# B&R Automation Studio project 8238 (part 9)

#### mnCntCyclic.st - Cyclic code
```iecst
(********************************************************************
 * COPYRIGHT -- Microsoft
 ********************************************************************
 * Program: mnCnt
 * File: mnCntCyclic.st
 * Author: hunholz
 * Created: July 02, 2011
 * Changed: January 3, 2012
 ********************************************************************
 * Implementation of program mnCnt
 ********************************************************************)

PROGRAM _CYCLIC

	/////////////
	// BATCHDATEN
	/////////////

	IF IFmnCnt.In.bBatchEventValid > 0 AND NOT IFmnCnt.Out.xBatchEventReadOK THEN

		// RB Eintrag
		// Jedes Batch-Event wird in den Ringbuffer eingetregen
		IF _xBatchRbOK AND IFmnCnt.In.BatchEvent.bEvent <= MNCNT_BATCHEVENT_DELETE THEN

			_rbBatchIns(pEntry := ADR(IFmnCnt.In.BatchEvent), wPtrWrite := _wPtrWriteBatch, wPtrRead := _wPtrReadBatch, wPtrStart := _wPtrStartBatch);

			IF _rbBatchIns.wStatus <> ERR_OK THEN

				_xBatchRbOK := FALSE;

			END_IF

		END_IF

		// Statistik ergänzen
		// Für jedes Entlade-Event wird ein Gesamtsummenzähler sowie ein Programm-Summenzähler gezählt
		IF _xBatchStatOK AND IFmnCnt.In.BatchEvent.bEvent = MNCNT_BATCHEVENT_UNLOAD THEN

			REPEAT

				_dwBatchStat.enable := TRUE;
				_dwBatchStat.ident := _doBatchStat.ident;
				_dwBatchStat.len := SIZEOF(_lSumWeight);
				_dwBatchStat.pSource := ADR(_lSumWeight);

				IF IFmnCnt.In.BatchEvent.bProgram <= 99 THEN

					// Zunächst die Zähler pro Programm addieren und in das Datenobjekt schreiben. Erst für den 1. Zähler, dann für den 2. Zähler
					_lSumWeight := _BatchStat.Weight1[IFmnCnt.In.BatchEvent.bProgram] + UINT_TO_UDINT(IFmnCnt.In.BatchEvent.Batch.wTotalWeight);

					_dwBatchStat.Offset := ADR(_BatchStat.Weight1[IFmnCnt.In.BatchEvent.bProgram]) - _doBatchStat.pDatObjMem;
					_dwBatchStat();

					IF _dwBatchStat.status <> ERR_OK THEN

						_xBatchStatOK := FALSE;

						EXIT;

					END_IF

					_lSumWeight := _BatchStat.Weight2[IFmnCnt.In.BatchEvent.bProgram] + UINT_TO_UDINT(IFmnCnt.In.BatchEvent.Batch.wTotalWeight);

					_dwBatchStat.Offset := ADR(_BatchStat.Weight2[IFmnCnt.In.BatchEvent.bProgram]) - _doBatchStat.pDatObjMem;
					_dwBatchStat();

					IF _dwBatchStat.status <> ERR_OK THEN

						_xBatchStatOK := FALSE;

						EXIT;

					END_IF

				END_IF

				// Dann wird der Gesamtzähler addiert

				_lSumWeight := _BatchStat.Weight1[100] + UINT_TO_UDINT(IFmnCnt.In.BatchEvent.Batch.wTotalWeight);

				_dwBatchStat.Offset := ADR(_BatchStat.Weight1[100]) - _doBatchStat.pDatObjMem;
				_dwBatchStat();

				IF _dwBatchStat.status <> ERR_OK THEN

					_xBatchStatOK := FALSE;

					EXIT;

				END_IF

				_lSumWeight := _BatchStat.Weight2[100] + UINT_TO_UDINT(IFmnCnt.In.BatchEvent.Batch.wTotalWeight);

				_dwBatchStat.Offset := ADR(_BatchStat.Weight2[100]) - _doBatchStat.pDatObjMem;
				_dwBatchStat();

				IF _dwBatchStat.status <> ERR_OK THEN

					_xBatchStatOK := FALSE;

					EXIT;

				END_IF

				UNTIL

				TRUE

			END_REPEAT

		END_IF

		IFmnCnt.Out.xBatchEventReadOK := _xBatchRbOK AND _xBatchStatOK;

	ELSIF IFmnCnt.In.bBatchEventValid = 0 THEN

		IFmnCnt.Out.xBatchEventReadOK := FALSE;

	END_IF

	//////////////
	// ZÄHLERDATEN
	//////////////

	FOR _i := 0 TO MNCNT_IDX_COUNTER_MAX DO

		IF IFmnCnt.In.bCntEventValid[_i] > 0 AND NOT IFmnCnt.Out.xCounterEventReadOK[_i] THEN

			// Ringbuffer Eintrag

			IF _xCounterRbOK THEN

				_rbCounterIns(pEntry := ADR(IFmnCnt.In.CounterEvent[_i]), wPtrWrite := _wPtrWriteCounter, wPtrRead := _wPtrReadCounter, wPtrStart := _wPtrStartCounter);

			END_IF

			IF _rbCounterIns.wStatus <> ERR_OK THEN

				_xCounterRbOK := FALSE;

			END_IF

			// Zählbare Zählerevents aufaddieren

			IF _xCounterStatOK AND IFmnCnt.In.CounterEvent[_i].lAmount > 0 AND IFmnCnt.In.CounterEvent[_i].bType < MNCNT_COUNTERTYPE_NOTCOUNTABLE THEN

				REPEAT

					// Zählernamen schreiben
					_dwCounterStat.enable := TRUE;
					_dwCounterStat.ident := _doCounterStat.ident;

					_dwCounterStat.pSource := ADR(IFmnCnt.In.CounterEvent[_i].Source.sNameId);
					_dwCounterStat.len := SIZEOF(_CounterStat.sCounterNameId[0]);
					_dwCounterStat.Offset := ADR(_CounterStat.sCounterNameId[_i]) - _doCounterStat.pDatObjMem;

					_dwCounterStat();

					IF _dwCounterStat.status <> ERR_OK THEN

						_xCounterStatOK := FALSE;

						EXIT;

					END_IF

					// Zählertyp schreiben
					_dwCounterStat.pSource := ADR(IFmnCnt.In.CounterEvent[_i].bType);
					_dwCounterStat.len := SIZEOF(_CounterStat.bCounterType[0]);
					_dwCounterStat.Offset := ADR(_CounterStat.bCounterType[_i]) - _doCounterStat.pDatObjMem;

					_dwCounterStat();

					IF _dwCounterStat.status <> ERR_OK THEN

						_xCounterStatOK := FALSE;

						EXIT;

					END_IF

					// Ersten Zähler addieren
					_lCounter := _CounterStat.Counter1[_i] + IFmnCnt.In.CounterEvent[_i].lAmount;

					_dwCounterStat.pSource := ADR(_lCounter);
					_dwCounterStat.len := SIZEOF(_CounterStat.Counter1[0]);
					_dwCounterStat.Offset := ADR(_CounterStat.Counter1[_i]) - _doCounterStat.pDatObjMem;

					_dwCounterStat();

					IF _dwCounterStat.status <> ERR_OK THEN

						_xCounterStatOK := FALSE;

						EXIT;

					END_IF

					// Zweiten Zähler addieren
					_lCounter := _CounterStat.Counter2[_i] + IFmnCnt.In.CounterEvent[_i].lAmount;

					_dwCounterStat.Offset := ADR(_CounterStat.Counter2[_i]) - _doCounterStat.pDatObjMem;

					_dwCounterStat();

					IF _dwCounterStat.status <> ERR_OK THEN

						_xCounterStatOK := FALSE;

						EXIT;

					END_IF

					UNTIL

					TRUE

				END_REPEAT

			END_IF

			IFmnCnt.Out.xCounterEventReadOK[_i] := _xCounterRbOK AND _xCounterStatOK;

		ELSIF IFmnCnt.In.bCntEventValid[_i] = 0 THEN

			IFmnCnt.Out.xCounterEventReadOK[_i] := FALSE;

		END_IF

	END_FOR

	//////////////
	// ZEITDATEN
	//////////////

	IF IFmnCnt.In.bTimeEventValid > 0 AND NOT IFmnCnt.Out.xTimeEventReadOK THEN

		// Ringbuffer Eintrag

		IF _xTimerRbOK THEN

			_rbTimerIns(pEntry := ADR(IFmnCnt.In.TimeEvent), wPtrWrite := _wPtrWriteTimer, wPtrRead := _wPtrReadTimer, wPtrStart := _wPtrStartTimer);

		END_IF

		IF _rbTimerIns.wStatus <> ERR_OK THEN

			_xTimerRbOK := FALSE;

		END_IF

		IF _xTimerStatOK AND IFmnCnt.In.TimeEvent.bState <= MNCNT_IDX_TIMESTATE_MAX AND IFmnCnt.In.TimeEvent.bSubState <= MNCNT_IDX_TIMESUBSTATE_MAX
			AND IFmnCnt.In.TimeEvent.lAmount > 0 THEN

			REPEAT

				_dwTimerStat.enable := TRUE;
				_dwTimerStat.ident := _doTimerStat.ident;

				// Ersten Zeitzähler addieren
				_lTime := _TimerStat.Counter1[IFmnCnt.In.TimeEvent.bState,IFmnCnt.In.TimeEvent.bSubState] + IFmnCnt.In.TimeEvent.lAmount;

				_dwTimerStat.pSource := ADR(_lTime);
				_dwTimerStat.len := SIZEOF(_TimerStat.Counter1[0,0]);
				_dwTimerStat.Offset := ADR(_TimerStat.Counter1[IFmnCnt.In.TimeEvent.bState,IFmnCnt.In.TimeEvent.bSubState]) - _doTimerStat.pDatObjMem;

				_dwTimerStat();

				IF _dwTimerStat.status <> ERR_OK THEN

					_xTimerStatOK := FALSE;

					EXIT;

				END_IF

				// Zweiten Zeitzähler addieren
				_lTime := _TimerStat.Counter2[IFmnCnt.In.TimeEvent.bState,IFmnCnt.In.TimeEvent.bSubState] + IFmnCnt.In.TimeEvent.lAmount;

				_dwTimerStat.Offset := ADR(_TimerStat.Counter2[IFmnCnt.In.TimeEvent.bState,IFmnCnt.In.TimeEvent.bSubState]) - _doTimerStat.pDatObjMem;

				_dwTimerStat();

				IF _dwTimerStat.status <> ERR_OK THEN

					_xTimerStatOK := FALSE;

					EXIT;

				END_IF

				UNTIL

				TRUE

			END_REPEAT

		END_IF

		IFmnCnt.Out.xTimeEventReadOK := _xTimerRbOK AND _xTimerStatOK;

	ELSIF IFmnCnt.In.bTimeEventValid = 0 THEN

		IFmnCnt.Out.xTimeEventReadOK := FALSE;

	END_IF

	//////////////
	// DOSIERDATEN
	//////////////

	FOR _i := 1 TO 48 DO

		IF IFmnCnt.In.bDosingEventValid[_i] > 0 AND NOT IFmnCnt.Out.xDosingEventReadOK[_i] THEN

			// Ringbuffer Eintrag

			IF _xDoseRbOK THEN

				_DosingEvent.DosingEvent := IFmnCnt.In.DosingEvent[_i];
				_DosingEvent.bId := UINT_TO_USINT(_i);
				_rbDoseIns(pEntry := ADR(_DosingEvent), wPtrWrite := _wPtrWriteDose, wPtrRead := _wPtrReadDose, wPtrStart := _wPtrStartDose);

			END_IF

			IF _rbDoseIns.wStatus <> ERR_OK THEN

				_xDoseRbOK := FALSE;

			END_IF

			IF _xDoseStatOK AND IFmnCnt.In.DosingEvent[_i].rAmount >= 0.001 THEN

				REPEAT

					_dwDosingStat.enable := TRUE;
					_dwDosingStat.ident := _doDosingStat.ident;

					// Namen der Dosierung schreiben
					_dwDosingStat.pSource := ADR(IFmnCnt.In.DosingEvent[_i].utfName);
					_dwDosingStat.len := SIZEOF(_DoseStat.utfDosingName[1]);
					_dwDosingStat.Offset := ADR(_DoseStat.utfDosingName[_i]) - _doDosingStat.pDatObjMem;

					_dwDosingStat();

					IF _dwDosingStat.status <> ERR_OK THEN

						_xDoseStatOK := FALSE;

						EXIT;

					END_IF

					// Einheit der Dosiermenge schreiben
					_dwDosingStat.pSource := ADR(IFmnCnt.In.DosingEvent[_i].sUnit);
					_dwDosingStat.len := SIZEOF(_DoseStat.sUnit[1]);
					_dwDosingStat.Offset := ADR(_DoseStat.sUnit[_i]) - _doDosingStat.pDatObjMem;

					_dwDosingStat();

					IF _dwDosingStat.status <> ERR_OK THEN

						_xDoseStatOK := FALSE;

						EXIT;

					END_IF

					// Pumpenkonstante schreiben
					_dwDosingStat.pSource := ADR(IFmnCnt.In.DosingEvent[_i].rPumpConst);
					_dwDosingStat.len := SIZEOF(_DoseStat.rPumpConst[1]);
					_dwDosingStat.Offset := ADR(_DoseStat.rPumpConst[_i]) - _doDosingStat.pDatObjMem;

					_dwDosingStat();

					IF _dwDosingStat.status <> ERR_OK THEN

						_xDoseStatOK := FALSE;

						EXIT;

					END_IF

					// Ersten Zähler für Dosiermenge addieren
					_rDoseingAmount := _DoseStat.Counter1[_i] + IFmnCnt.In.DosingEvent[_i].rAmount;

					_dwDosingStat.pSource := ADR(_rDoseingAmount);
					_dwDosingStat.len := SIZEOF(_DoseStat.Counter1[1]);
					_dwDosingStat.Offset := ADR(_DoseStat.Counter1[_i]) - _doDosingStat.pDatObjMem;

					_dwDosingStat();

					IF _dwDosingStat.status <> ERR_OK THEN

						_xDoseStatOK := FALSE;

						EXIT;

					END_IF

					// Zweiten Zähler für Dosiermenge addieren
					_rDoseingAmount := _DoseStat.Counter2[_i] + IFmnCnt.In.DosingEvent[_i].rAmount;

					_dwDosingStat.Offset := ADR(_DoseStat.Counter2[_i]) - _doDosingStat.pDatObjMem;

					_dwDosingStat();

					IF _dwDosingStat.status <> ERR_OK THEN

						_xDoseStatOK := FALSE;

						EXIT;

					END_IF

					UNTIL

					TRUE

				END_REPEAT

			END_IF

			IFmnCnt.Out.xDosingEventReadOK[_i] := _xDoseRbOK AND _xDoseStatOK;

		ELSIF IFmnCnt.In.bDosingEventValid[_i] = 0 THEN

			IFmnCnt.Out.xDosingEventReadOK[_i] := FALSE;

		END_IF

	END_FOR

	// Batchdaten an hlDFII senden

	// Senden nach 5 Sekunden wiederholen, wenn die letzte Sendung fehlerhaft war
	_TONrepeatDFIIBatchEvt(IN := (IFhlDFII.Out.RespCntBatchEvt.wResponse <> ERR_FUB_BUSY) AND (IFhlDFII.Out.RespCntBatchEvt.wResponse <> 0)
			AND (IFhlDFII.Out.RespCntBatchEvt.wResponse <> IFhlDFII.In.ReqCntBatchEvt.wRequest), PT := T#5s);

	IF _xBatchRbOK THEN

		IF IFhlDFII.Out.RespCntBatchEvt.wResponse = 0 AND IFhlDFII.In.ReqCntBatchEvt.wRequest = 0 THEN

			// Die Schnittstelle zur Datenbank ist bereit!

			IF NOT _xRepeatDFIIBatchEvt THEN

				// Daten nur dann aus dem Ringbuffer lesen, wenn nicht wiederholt werden soll.

				IFhlDFII.In.ReqCntBatchEvt.bCntLines := 0;

				FOR _ii := 0 TO 4 DO

					_rbBatchRead(wPtrWrite := _wPtrWriteBatch, pEntry := ADR(IFhlDFII.In.ReqCntBatchEvt.CntBatchEvtList[_ii+1]), wPtrStart := _wPtrStartBatch, wPtrRead := _wPtrReadBatch);

					IF _rbBatchRead.wStatus <> 0 THEN
						// Ringbuffer hat keinen neuen Eintrag
						EXIT;
					END_IF

					IFhlDFII.In.ReqCntBatchEvt.bCntLines := IFhlDFII.In.ReqCntBatchEvt.bCntLines + 1;

				END_FOR

			END_IF

			_xRepeatDFIIBatchEvt := FALSE;

			IF IFhlDFII.In.ReqCntBatchEvt.bCntLines > 0 THEN
				// Senden wird nur ausgelöst, wenn der Ringbuffer einen neuen Eintrag hatte.
				IFhlDFII.In.ReqCntBatchEvt.wRequest := 1;

			END_IF

		ELSIF IFhlDFII.Out.RespCntBatchEvt.wResponse = IFhlDFII.In.ReqCntBatchEvt.wRequest THEN

			IFhlDFII.In.ReqCntBatchEvt.wRequest := 0;

		ELSIF IFhlDFII.Out.RespCntBatchEvt.wResponse <> ERR_FUB_BUSY AND _TONrepeatDFIIBatchEvt.Q THEN

			IFhlDFII.In.ReqCntBatchEvt.wRequest := 0;

			_xRepeatDFIIBatchEvt := TRUE;

		END_IF

	END_IF

	// Counter-Daten an hlDFII senden

	// Senden nach 5 Sekunden wiederholen, wenn die letzte Sendung fehlerhaft war
	_TONrepeatDFIICounterEvt(IN := (IFhlDFII.Out.RespCntCntEvt.wResponse <> ERR_FUB_BUSY) AND (IFhlDFII.Out.RespCntCntEvt.wResponse <> 0)
	AND (IFhlDFII.Out.RespCntCntEvt.wResponse <> IFhlDFII.In.ReqCntCntEvt.wRequest), PT := T#5s);

	IF _xCounterRbOK THEN

		IF IFhlDFII.Out.RespCntCntEvt.wResponse = 0 AND IFhlDFII.In.ReqCntCntEvt.wRequest = 0 THEN

			// Die Schnittstelle zur Datenbank ist bereit!

			IF NOT _xRepeatDFIICounterEvt THEN

				// Daten nur dann aus dem Ringbuffer lesen, wenn nicht wiederholt werden soll.

				IFhlDFII.In.ReqCntCntEvt.bCntLines := 0;

				FOR _ii := 0 TO 4 DO

					_rbCounterRead(wPtrWrite := _wPtrWriteCounter, pEntry := ADR(IFhlDFII.In.ReqCntCntEvt.CntCounterEvtList[_ii+1]), wPtrStart := _wPtrStartCounter, wPtrRead := _wPtrReadCounter);

					IF _rbCounterRead.wStatus <> 0 THEN
						// Ringbuffer hat keinen neuen Eintrag
						EXIT;
					END_IF

					IFhlDFII.In.ReqCntCntEvt.bCntLines := IFhlDFII.In.ReqCntCntEvt.bCntLines + 1;

				END_FOR

			END_IF

			_xRepeatDFIICounterEvt := FALSE;

			IF IFhlDFII.In.ReqCntCntEvt.bCntLines > 0 THEN
				// Senden wird nur ausgelöst, wenn der Ringbuffer einen neuen Eintrag hatte.
				IFhlDFII.In.ReqCntCntEvt.wRequest := 1;

			END_IF

		ELSIF IFhlDFII.Out.RespCntCntEvt.wResponse = IFhlDFII.In.ReqCntCntEvt.wRequest THEN

			IFhlDFII.In.ReqCntCntEvt.wRequest := 0;

		ELSIF IFhlDFII.Out.RespCntCntEvt.wResponse <> ERR_FUB_BUSY AND _TONrepeatDFIICounterEvt.Q THEN

			IFhlDFII.In.ReqCntCntEvt.wRequest := 0;

			_xRepeatDFIICounterEvt := TRUE;

		END_IF

	END_IF

	// Timer-Daten an hlDFII senden

	// Senden nach 5 Sekunden wiederholen, wenn die letzte Sendung fehlerhaft war
	_TONrepeatDFIITimerEvt(IN := (IFhlDFII.Out.RespCntTimEvt.wResponse <> ERR_FUB_BUSY) AND (IFhlDFII.Out.RespCntTimEvt.wResponse <> 0)
	AND (IFhlDFII.Out.RespCntTimEvt.wResponse <> IFhlDFII.In.ReqCntTimEvt.wRequest), PT := T#5s);

	IF _xTimerRbOK THEN

		IF IFhlDFII.Out.RespCntTimEvt.wResponse = 0 AND IFhlDFII.In.ReqCntTimEvt.wRequest = 0 THEN

			// Die Schnittstelle zur Datenbank ist bereit!

			IF NOT _xRepeatDFIITimerEvt THEN

				// Daten nur dann aus dem Ringbuffer lesen, wenn nicht wiederholt werden soll.

				IFhlDFII.In.ReqCntTimEvt.bCntLines := 0;

				FOR _ii := 0 TO 4 DO

					_rbTimerRead(wPtrWrite := _wPtrWriteTimer, pEntry := ADR(IFhlDFII.In.ReqCntTimEvt.CntTimerEvtList[_ii+1]), wPtrStart := _wPtrStartTimer, wPtrRead := _wPtrReadTimer);

					IF _rbTimerRead.wStatus <> 0 THEN
						// Ringbuffer hat keinen neuen Eintrag
						EXIT;
					END_IF

					IFhlDFII.In.ReqCntTimEvt.bCntLines := IFhlDFII.In.ReqCntTimEvt.bCntLines + 1;

				END_FOR

			END_IF

			_xRepeatDFIITimerEvt := FALSE;

			IF IFhlDFII.In.ReqCntTimEvt.bCntLines > 0 THEN
				// Senden wird nur ausgelöst, wenn der Ringbuffer einen neuen Eintrag hatte.
				IFhlDFII.In.ReqCntTimEvt.wRequest := 1;

			END_IF

		ELSIF IFhlDFII.Out.RespCntTimEvt.wResponse = IFhlDFII.In.ReqCntTimEvt.wRequest THEN

			IFhlDFII.In.ReqCntTimEvt.wRequest := 0;

		ELSIF IFhlDFII.Out.RespCntTimEvt.wResponse <> ERR_FUB_BUSY AND _TONrepeatDFIITimerEvt.Q THEN

			IFhlDFII.In.ReqCntTimEvt.wRequest := 0;

			_xRepeatDFIITimerEvt := TRUE;

		END_IF

	END_IF

	// Dosing-Daten an hlDFII senden

	// Senden nach 5 Sekunden wiederholen, wenn die letzte Sendung fehlerhaft war
	_TONrepeatDFIIDoseEvt(IN := (IFhlDFII.Out.RespCntDosEvt.wResponse <> ERR_FUB_BUSY) AND (IFhlDFII.Out.RespCntDosEvt.wResponse <> 0)
	AND (IFhlDFII.Out.RespCntDosEvt.wResponse <> IFhlDFII.In.ReqCntDosEvt.wRequest), PT := T#5s);

	IF _xDoseRbOK THEN

		IF IFhlDFII.Out.RespCntDosEvt.wResponse = 0 AND IFhlDFII.In.ReqCntDosEvt.wRequest = 0 THEN

			// Die Schnittstelle zur Datenbank ist bereit!

			IF NOT _xRepeatDFIIDoseEvt THEN

				// Daten nur dann aus dem Ringbuffer lesen, wenn nicht wiederholt werden soll.

				IFhlDFII.In.ReqCntDosEvt.bCntLines := 0;

				FOR _ii := 0 TO 4 DO

					_rbDoseRead(wPtrWrite := _wPtrWriteDose, pEntry := ADR(IFhlDFII.In.ReqCntDosEvt.CntDosingEvtList[_ii+1]), wPtrStart := _wPtrStartDose, wPtrRead := _wPtrReadDose);

					IF _rbDoseRead.wStatus <> 0 THEN
						// Ringbuffer hat keinen neuen Eintrag
						EXIT;
					END_IF

					IFhlDFII.In.ReqCntDosEvt.bCntLines := IFhlDFII.In.ReqCntDosEvt.bCntLines + 1;

				END_FOR

			END_IF

			_xRepeatDFIIDoseEvt := FALSE;

			IF IFhlDFII.In.ReqCntDosEvt.bCntLines > 0 THEN
				// Senden wird nur ausgelöst, wenn der Ringbuffer einen neuen Eintrag hatte.
				IFhlDFII.In.ReqCntDosEvt.wRequest := 1;

			END_IF

		ELSIF IFhlDFII.Out.RespCntDosEvt.wResponse = IFhlDFII.In.ReqCntDosEvt.wRequest THEN

			IFhlDFII.In.ReqCntDosEvt.wRequest := 0;

		ELSIF IFhlDFII.Out.RespCntDosEvt.wResponse <> ERR_FUB_BUSY AND _TONrepeatDFIIDoseEvt.Q THEN

			IFhlDFII.In.ReqCntDosEvt.wRequest := 0;

			_xRepeatDFIIDoseEvt := TRUE;

		END_IF

	END_IF

END_PROGRAM
```

#### mnCntInit.st - Initialization code
```iecst
(********************************************************************
 * COPYRIGHT -- Microsoft
 ********************************************************************
 * Program: mnCnt
 * File: mnCntInit.st
 * Author: hunholz
 * Created: July 02, 2011
 ********************************************************************
 * Implementation of program mnCnt
 ********************************************************************)

PROGRAM _INIT

	// Packet-Version auslesen mit MO_ver aus SYS_lib und für den Additional Status zur Verfügung stellen

	_sPkgName := 'mnCnt';

	IF ( MO_ver(ADR(_sPkgName), 0, ADR(_VerStruc)) = 0 ) THEN

		brsmemcpy(ADR(mnCntStatAd.sPkgVersion), ADR(_VerStruc.version), SIZEOF(_VerStruc.version));

	ELSE

		mnCntStatAd.sPkgVersion := '---';

	END_IF

	// Initialisierungen

	// Function ID von mnCnt
	kgMsgStatus[MNCNT_IDX_KGMSGSTAT].wFunction_ID := 6;

	// =============
	// Batche-Events
	// =============

	IFmnCnt.Out.xBatchEventReadOK := FALSE;

	// Statistik prüfen

	_doBatchStat.enable := TRUE;
	_doBatchStat.pName := ADR(_DataObjectName.sBatchStatName);
	_doBatchStat();

	IF _doBatchStat.status <> ERR_OK THEN

		_dcBatchStat.enable := TRUE;
		_dcBatchStat.MemType := doUSRROM;
		_dcBatchStat.pName := ADR(_DataObjectName.sBatchStatName);
		_dcBatchStat.len := SIZEOF(_BatchStat);
		_dcBatchStat();

		_doBatchStat();

	END_IF

	IF _doBatchStat.status = ERR_OK THEN

		_BatchStat ACCESS _doBatchStat.pDatObjMem;

		_xBatchStatOK := TRUE;

	END_IF

	// Ringbuffer prüfen

	_kgRBcreateBatch.sName := _DataObjectName.sBatchRBName;
	_kgRBcreateBatch.bMemType := doUSRROM;
	_kgRBcreateBatch.lLenEntry := SIZEOF(_BatchRB[1]);
	_kgRBcreateBatch.wCntEntry := MNCNT_MAX_RBENTRY_BATCH;

	_kgRBcreateBatch(wPtrWrite := _wPtrWriteBatch , wPtrRead := _wPtrReadBatch, wPtrStart := _wPtrStartBatch);

	IF _kgRBcreateBatch.wStatus = ERR_OK THEN

		_rbBatchIns.doIdent 	:= _kgRBcreateBatch.doIdent;
		_rbBatchIns.doLen		:= _kgRBcreateBatch.doLen;
		_rbBatchIns.lLenEntry	:= SIZEOF(_BatchRB[1]);

		_rbBatchRead.doIdent 	:= _kgRBcreateBatch.doIdent;
		_rbBatchRead.doLen		:= _kgRBcreateBatch.doLen;
		_rbBatchRead.lLenEntry	:= SIZEOF(_BatchRB[1]);

		_xBatchRbOK 			:= TRUE;

		_BatchRB ACCESS _kgRBcreateBatch.pDatObjMem;

	END_IF

	// =============
	// Counter-Events
	// =============

	brsmemset(ADR(IFmnCnt.Out.xCounterEventReadOK), 0, SIZEOF(IFmnCnt.Out.xCounterEventReadOK));

	// Statistik prüfen

	_doCounterStat.enable := TRUE;
	_doCounterStat.pName := ADR(_DataObjectName.sCountStatName);
	_doCounterStat();

	IF _doCounterStat.status = ERR_OK THEN

		// Statistik wurde vergrößtert, d.h. die aktuelle wird gelöscht
		IF _doCounterStat.len < SIZEOF(_CounterStat) THEN

			_ddCounterStat.enable := TRUE;
			_ddCounterStat.ident := _doCounterStat.ident;
			_ddCounterStat();

			_doCounterStat();

		END_IF

	END_IF

	IF _doCounterStat.status <> ERR_OK THEN

		_dcCounterStat.enable := TRUE;
		_dcCounterStat.MemType := doUSRROM;
		_dcCounterStat.pName := ADR(_DataObjectName.sCountStatName);
		_dcCounterStat.len := SIZEOF(_CounterStat);
		_dcCounterStat();

		_doCounterStat();

	END_IF

	IF _doCounterStat.status = ERR_OK THEN

		_CounterStat ACCESS _doCounterStat.pDatObjMem;

		_xCounterStatOK := TRUE;

	END_IF

	// Ringbuffer prüfen

	_kgRBcreateCounter.sName := _DataObjectName.sCountRBName;
	_kgRBcreateCounter.bMemType := doUSRROM;
	_kgRBcreateCounter.lLenEntry := SIZEOF(_CounterRB[1]);
	_kgRBcreateCounter.wCntEntry := MNCNT_MAX_RBENTRY_COUNTER;

	_kgRBcreateCounter(wPtrWrite := _wPtrWriteCounter , wPtrRead := _wPtrReadCounter, wPtrStart := _wPtrStartCounter);

	IF _kgRBcreateCounter.wStatus = ERR_OK THEN

		_rbCounterIns.doIdent 	:= _kgRBcreateCounter.doIdent;
		_rbCounterIns.doLen		:= _kgRBcreateCounter.doLen;
		_rbCounterIns.lLenEntry	:= SIZEOF(_CounterRB[1]);

		_rbCounterRead.doIdent 	:= _kgRBcreateCounter.doIdent;
		_rbCounterRead.doLen		:= _kgRBcreateCounter.doLen;
		_rbCounterRead.lLenEntry	:= SIZEOF(_CounterRB[1]);

		_xCounterRbOK 			:= TRUE;

		_CounterRB ACCESS _kgRBcreateCounter.pDatObjMem;

	END_IF

	// =============
	// Timer-Events
	// =============

	brsmemset(ADR(IFmnCnt.Out.xTimeEventReadOK), 0, SIZEOF(IFmnCnt.Out.xTimeEventReadOK));

	// Statistik prüfen

	_doTimerStat.enable := TRUE;
	_doTimerStat.pName := ADR(_DataObjectName.sTimeStatName);
	_doTimerStat();

	IF _doTimerStat.status = ERR_OK THEN

		// Statistik wurde vergrößtert, d.h. die aktuelle wird gelöscht
		IF _doTimerStat.len < SIZEOF(_TimerStat) THEN

			_ddTimerStat.enable := TRUE;
			_ddTimerStat.ident := _doTimerStat.ident;
			_ddTimerStat();

			_doTimerStat();

		END_IF

	END_IF

	IF _doTimerStat.status <> ERR_OK THEN

		_dcTimerStat.enable := TRUE;
		_dcTimerStat.MemType := doUSRROM;
		_dcTimerStat.pName := ADR(_DataObjectName.sTimeStatName);
		_dcTimerStat.len := SIZEOF(_TimerStat);
		_dcTimerStat();

		_doTimerStat();

	END_IF

	IF _doTimerStat.status = ERR_OK THEN

		_TimerStat ACCESS _doTimerStat.pDatObjMem;

		_xTimerStatOK := TRUE;

	END_IF

	// Ringbuffer prüfen

	_kgRBcreateTimer.sName := _DataObjectName.sTimeRBName;
	_kgRBcreateTimer.bMemType := doUSRROM;
	_kgRBcreateTimer.lLenEntry := SIZEOF(_TimerRB[1]);
	_kgRBcreateTimer.wCntEntry := MNCNT_MAX_RBENTRY_TIME;

	_kgRBcreateTimer(wPtrWrite := _wPtrWriteTimer , wPtrRead := _wPtrReadTimer, wPtrStart := _wPtrStartTimer);

	IF _kgRBcreateTimer.wStatus = ERR_OK THEN

		_rbTimerIns.doIdent 	:= _kgRBcreateTimer.doIdent;
		_rbTimerIns.doLen		:= _kgRBcreateTimer.doLen;
		_rbTimerIns.lLenEntry	:= SIZEOF(_TimerRB[1]);

		_rbTimerRead.doIdent 	:= _kgRBcreateTimer.doIdent;
		_rbTimerRead.doLen		:= _kgRBcreateTimer.doLen;
		_rbTimerRead.lLenEntry	:= SIZEOF(_TimerRB[1]);

		_xTimerRbOK 			:= TRUE;

		_TimerRB ACCESS _kgRBcreateTimer.pDatObjMem;

	END_IF

	// =============
	// Dosing-Events
	// =============

	brsmemset(ADR(IFmnCnt.Out.xDosingEventReadOK), 0, SIZEOF(IFmnCnt.Out.xDosingEventReadOK));

	// Statistik prüfen

	_doDosingStat.enable := TRUE;
	_doDosingStat.pName := ADR(_DataObjectName.sDoseStatName);
	_doDosingStat();

	IF _doDosingStat.status = ERR_OK THEN

		// Statistik wurde vergrößtert, d.h. die aktuelle wird gelöscht
		IF _doDosingStat.len < SIZEOF(_DoseStat) THEN

			_ddDosingStat.enable := TRUE;
			_ddDosingStat.ident := _doDosingStat.ident;
			_ddDosingStat();

			_doDosingStat();

		END_IF

	END_IF

	IF _doDosingStat.status <> ERR_OK THEN

		_dcDosingStat.enable := TRUE;
		_dcDosingStat.MemType := doUSRROM;
		_dcDosingStat.pName := ADR(_DataObjectName.sDoseStatName);
		_dcDosingStat.len := SIZEOF(_DoseStat);
		_dcDosingStat();

		_doDosingStat();

	END_IF

	IF _doDosingStat.status = ERR_OK THEN

		_DoseStat ACCESS _doDosingStat.pDatObjMem;

		_xDoseStatOK := TRUE;

	END_IF

	// Ringbuffer prüfen

	_kgRBcreateDosing.sName := _DataObjectName.sDoseRBName;
	_kgRBcreateDosing.bMemType := doUSRROM;
	_kgRBcreateDosing.lLenEntry := SIZEOF(_DoseRB[1]);
	_kgRBcreateDosing.wCntEntry := MNCNT_MAX_RBENTRY_DOSE;

	_kgRBcreateDosing(wPtrWrite := _wPtrWriteDose , wPtrRead := _wPtrReadDose, wPtrStart := _wPtrStartDose);

	IF _kgRBcreateDosing.wStatus = ERR_OK THEN

		_rbDoseIns.doIdent 	:= _kgRBcreateDosing.doIdent;
		_rbDoseIns.doLen		:= _kgRBcreateDosing.doLen;
		_rbDoseIns.lLenEntry	:= SIZEOF(_DoseRB[1]);

		_rbDoseRead.doIdent 	:= _kgRBcreateDosing.doIdent;
		_rbDoseRead.doLen		:= _kgRBcreateDosing.doLen;
		_rbDoseRead.lLenEntry	:= SIZEOF(_DoseRB[1]);

		_xDoseRbOK 			:= TRUE;

		_DoseRB ACCESS _kgRBcreateDosing.pDatObjMem;

	END_IF

END_PROGRAM
```

#### mnCnt.typ - Local data types
```iecst
(********************************************************************
 * COPYRIGHT -- Microsoft
 ********************************************************************
 * Program: mnCnt
 * File: mnCnt.typ
 * Author: hunholz
 * Created: November 11, 2011
 ********************************************************************
 * Local data types of program mnCnt
 ********************************************************************)

TYPE
	EventSumDel_enum :
		(
		Del_Delete,
		Del_Wait,
		Del_Create,
		Del_Info,
		Del_Write,
		Del_Error
		);
	mnCnt_BatchStat_typ : 	STRUCT
		Weight1 : ARRAY[0..100]OF UDINT;
		Weight2 : ARRAY[0..100]OF UDINT;
	END_STRUCT;
	mnCnt_CounterStat_typ : 	STRUCT
		sCounterNameId : ARRAY[0..MNCNT_IDX_COUNTER_MAX]OF STRING[10];
		bCounterType : ARRAY[0..MNCNT_IDX_COUNTER_MAX]OF USINT;
		Counter1 : ARRAY[0..MNCNT_IDX_COUNTER_MAX]OF UDINT;
		Counter2 : ARRAY[0..MNCNT_IDX_COUNTER_MAX]OF UDINT;
	END_STRUCT;
	mnCnt_TimerStat_typ : 	STRUCT
		Counter1 : ARRAY[0..MNCNT_IDX_TIMESTATE_MAX,0..MNCNT_IDX_TIMESUBSTATE_MAX]OF UDINT;
		Counter2 : ARRAY[0..MNCNT_IDX_TIMESTATE_MAX,0..MNCNT_IDX_TIMESUBSTATE_MAX]OF UDINT;
	END_STRUCT;
	mnCnt_DoseStat_typ : 	STRUCT
		utfDosingName : ARRAY[1..48]OF WSTRING[23];
		sUnit : ARRAY[1..48]OF STRING[11];
		rPumpConst : ARRAY[1..48]OF REAL;
		Counter1 : ARRAY[1..48]OF REAL;
		Counter2 : ARRAY[1..48]OF REAL;
	END_STRUCT;
	mnCnt_DatObjNames_typ : 	STRUCT
		sBatchStatName : STRING[11] := '_mnCntBst';
		sBatchRBName : STRING[11] := '_mnCntBrb';
		sCountStatName : STRING[11] := '_mnCntCst';
		sCountRBName : STRING[11] := '_mnCntCrb';
		sTimeStatName : STRING[11] := '_mnCntTst';
		sTimeRBName : STRING[11] := '_mnCntTrb';
		sDoseStatName : STRING[11] := '_mnCntDst';
		sDoseRBName : STRING[11] := '_mnCntDrb';
	END_STRUCT;
END_TYPE
```

#### mnCnt.var - Local variables
```iecst
(********************************************************************
 * COPYRIGHT -- Microsoft
 ********************************************************************
 * Program: mnCnt
 * File: mnCnt.var
 * Author: hunholz
 * Created: November 11, 2011
 ********************************************************************
 * Local variables of program mnCnt
 ********************************************************************)
VAR
	_sPkgName : STRING[11];
	_VerStruc : MoVerStruc_typ;
END_VAR
(*Datenobjekte zum Speichern der Statistik und der Event-Ringbuffer*)
VAR
	_DataObjectName : mnCnt_DatObjNames_typ;
	_doBatchStat : DatObjInfo;
	_dcBatchStat : DatObjCreate;
	_dwBatchStat : DatObjWrite;
	_doCounterStat : DatObjInfo;
	_ddCounterStat : DatObjDelete;
	_dcCounterStat : DatObjCreate;
	_dwCounterStat : DatObjWrite;
	_doTimerStat : DatObjInfo;
	_ddTimerStat : DatObjDelete;
	_dcTimerStat : DatObjCreate;
	_dwTimerStat : DatObjWrite;
	_doDosingStat : DatObjInfo;
	_ddDosingStat : DatObjDelete;
	_dcDosingStat : DatObjCreate;
	_dwDosingStat : DatObjWrite;
END_VAR
(*Zeiger auf Statistiken*)
VAR
	_BatchStat : REFERENCE TO mnCnt_BatchStat_typ;
	_CounterStat : REFERENCE TO mnCnt_CounterStat_typ;
	_TimerStat : REFERENCE TO mnCnt_TimerStat_typ;
	_DoseStat : REFERENCE TO mnCnt_DoseStat_typ;
END_VAR
(*Zeiger auf Ringbuffer*)
VAR
	_BatchRB : REFERENCE TO ARRAY[1..MNCNT_MAX_RBENTRY_BATCH] OF mnCntEventBatch_Typ;
	_CounterRB : REFERENCE TO ARRAY[1..MNCNT_MAX_RBENTRY_COUNTER] OF mnCntEventCounter_Typ;
	_TimerRB : REFERENCE TO ARRAY[1..MNCNT_MAX_RBENTRY_TIME] OF mnCntEventTime_Typ;
	_DoseRB : REFERENCE TO ARRAY[1..MNCNT_MAX_RBENTRY_DOSE] OF mnCntEventDosingId_Typ;
END_VAR
(*Status von Statistiken und Ringbuffern*)
VAR
	_xBatchStatOK : BOOL;
	_xBatchRbOK : BOOL;
	_xCounterStatOK : BOOL;
	_xCounterRbOK : BOOL;
	_xTimerStatOK : BOOL;
	_xTimerRbOK : BOOL;
	_xDoseStatOK : BOOL;
	_xDoseRbOK : BOOL;
END_VAR
(*Ringbuffer Batch*)
VAR
	_kgRBcreateBatch : kgRBcreate;
	_rbBatchIns : kgRBinsert;
	_rbBatchRead : kgRBread;
END_VAR
VAR RETAIN
	_wPtrWriteBatch : UINT;
	_wPtrReadBatch : UINT;
	_wPtrStartBatch : UINT;
END_VAR
(*Ringbuffer Counter*)
VAR RETAIN
	_wPtrReadCounter : UINT := 0;
	_wPtrWriteCounter : UINT;
	_wPtrStartCounter : UINT;
END_VAR
VAR
	_kgRBcreateCounter : kgRBcreate;
	_rbCounterIns : kgRBinsert;
	_rbCounterRead : kgRBread;
END_VAR
(*Ringbuffer Timer*)
VAR RETAIN
	_wPtrReadTimer : UINT;
	_wPtrWriteTimer : UINT;
	_wPtrStartTimer : UINT;
END_VAR
VAR
	_kgRBcreateTimer : kgRBcreate;
	_rbTimerIns : kgRBinsert;
	_rbTimerRead : kgRBread;
END_VAR
(*Ringbuffer Dosing*)
VAR RETAIN
	_wPtrReadDose : UINT;
	_wPtrWriteDose : UINT;
	_wPtrStartDose : UINT;
END_VAR
VAR
	_kgRBcreateDosing : kgRBcreate;
	_rbDoseIns : kgRBinsert;
	_rbDoseRead : kgRBread;
END_VAR
(*Hilfsvariablen*)
VAR
	_i : UINT;
	_lSumWeight : UDINT;
	_lCounter : UDINT;
	_lTime : UDINT;
	_rDoseingAmount : REAL;
	_TONrepeatDFIIBatchEvt : TON;
	_xRepeatDFIIBatchEvt : BOOL;
	_ii : UINT;
	_DosingEvent : mnCntEventDosingId_Typ;
	_TONrepeatDFIICounterEvt : TON;
	_xRepeatDFIICounterEvt : BOOL;
	_TONrepeatDFIITimerEvt : TON;
	_xRepeatDFIITimerEvt : BOOL;
	_xRepeatDFIIDoseEvt : BOOL;
	_TONrepeatDFIIDoseEvt : TON;
END_VAR
```

### mnCnt-History.txt
```
0.12.0		09.01.2012	AH	- Version wird in mnCntStatAdd eingetragen.
							- Statistik verwalten, Ringbuffer verwalten, Daten an DFII senden
0.13.0		25.01.2012	AH Anpassung an KGStandard 1.13.0 (Ringbuffer)

0.14.0		26.01.2012  AH Substatus für Active erweitert. Prepforstop
0.14.1		07.02.2012	AH Startpointer wurde an RBread nicht übergeben. Damit kam es immer zum Status = 4
0.15.0		10.02.2012	AH Batcheven um zweite Location erweitert. CompNo im Location entfällt.
0.16.0		13.02.2012  AH Strukturänderungen in den Events. Fehlerbehebung beim Eintragen in die Requests an DFII
						   Kompatibel zu hlDFII 1.12.0
0.16.1		20.03.2012	AH Abhängigkeiten ergänzt
```

### Package Logical/Standard/Kanlink/KGFramework/Pkg_mnMsg - Meldungs-Manager

### Pkg_mnMsg.typ - Package data types
```iecst
(********************************************************************
 * COPYRIGHT -- Microsoft
 ********************************************************************
 * Package: Pkg_mnMsg
 * File: Pkg_mnMsg.typ
 * Author: hunholz/ subramaniam
 * Created: January 05, 2011
 * Changed: June 15, 2011
 ********************************************************************
 * Data types of package Pkg_mnMsg
 ********************************************************************)
(*Typdeklaration für kgMsgStat*)

TYPE
	kgMsg_Status_Typ : 	STRUCT
		wFunction_ID : UINT;
		wMsgClass : UINT;
		wMsgNumber : UINT;
		wMsgAckLevel : UINT;
		wInstance : UINT;
		sMsgAttrTxt : STRING[13];
		diMsgAttr1 : DINT;
		diMsgAttr2 : DINT;
		wMaintNumber : UINT;
		sMaintAttrTxt : STRING[13];
		diMaintAttr1 : DINT;
		diMaintAttr2 : DINT;
		wMaintAckLevel : UINT;
		xAckMaint : BOOL;
		xAckFault : BOOL;
		xAckAva : BOOL;
		xAckRead : BOOL;
	END_STRUCT;
END_TYPE

(*Konfigurationsstruktur *)

TYPE
	CfgMsgStatList_Typ : 	STRUCT
		wFunction_ID : UINT;
		wMsgNumber : UINT;
		wInstance : UINT;
		wRes : UINT;
	END_STRUCT;
END_TYPE

(*Struktur Meldungsstatistik *)

TYPE
	MsgStat_Typ : 	STRUCT
		Header : MsgStatHeader_Typ;
		List : ARRAY[1..MNMSG_MAX_CFGMESSAGES]OF MsgStatList_Typ;
	END_STRUCT;
	MsgStatHeader_Typ : 	STRUCT
		lVersion : UDINT;
		lLength : UDINT;
	END_STRUCT;
	MsgStatList_Typ : 	STRUCT
		wFunction_ID : UINT;
		wMsgNumber : UINT;
		wInstance : UINT;
		wMsgClass : UINT;
		lCnt : UDINT;
		lTime : UDINT;
	END_STRUCT;
END_TYPE

(*Synchrones (Internes) Interface zur Steuerung*)

TYPE
	IFmnMsgOutMsgList_Typ : 	STRUCT
		utfMsgText : WSTRING[67]; (*Meldungs-ID, Meldungs-Text*)
		utfMsgHelpText : WSTRING[255];
		wFunction_ID : UINT; (*Funktions-ID der Meldung*)
		wMsgNumber : UINT; (*Meldungs- oder Wartungsnummer*)
		bInstance : USINT; (*MeldungsInstanz*)
		bMsgClass : USINT; (*0..9 - Störung, 10..19 - Warnung, Info, 20 - Wartung*)
		bAckLevel : UINT; (*0 - jeder, 1 - Operator, 2 - Techniker, 3 - KG-Techniker, 4 - Admin, 255 - nicht quittierbar*)
	END_STRUCT;
	IFmnMsgOutMsgHistList_Typ : 	STRUCT
		utfMsgText : WSTRING[67]; (*Timestamp, Meldungs-ID, Meldungs-Text*)
		bMsgClass : USINT; (*0..9 - Störung, 10..19 - Warnung, Info, 20 - Wartung*)
		bEvent : USINT; (*1 - gekommen, 2 - quittiert, 3 - gegangen*)
	END_STRUCT;
	IFmnMsgOutMsgStatistic_Typ : 	STRUCT
		utfMsgText : WSTRING[67]; (*Meldungs-ID, Meldungs-Text*)
		lValue : UDINT; (*Anzahl der Meldungen bzw. Zeit der Meldungen*)
	END_STRUCT;
	IFmnMsgOut_Typ : 	STRUCT
		MsgList : ARRAY[0..MNMSG_MAX_IDX_VCMSGLIST]OF IFmnMsgOutMsgList_Typ; (*Meldungsliste zur lokalen Anzeige auf der SPS*)
		MsgHistList : ARRAY[0..MNMSG_MAX_IDX_VCMSGHISTLIST]OF IFmnMsgOutMsgHistList_Typ; (*Ausschnitt aus der Meldungshistorie*)
		MsgStatistic : ARRAY[0..MNMSG_MAX_IDX_VCMSGSTATLIST]OF IFmnMsgOutMsgStatistic_Typ;
		wMsgListCnt : UINT; (*Anzahl Meldungen in der Meldungsliste*)
		wMsgHistListCnt : UINT; (*Anzahl der Events in der historischen Meldungsliste*)
		wMsgHistListMaxOffset : UINT; (*Maximal möglicher Offset im Ringbuffer, d.h. Anzahl der Einträge im RB - 1 oder 0, wenn RB leer*)
		wMsgHistListOffset : UINT;
		wMsgStatisticCnt : UINT;
		xFaultInt : BOOL;
		xFaultExt : BOOL;
		xWarning : BOOL;
		xInformation : BOOL;
		xFault : BOOL;
		xReserve : BOOL;
		xMaintenance : BOOL;
		xMnMsgReady : BOOL;
		wCntFaultNoAck : UINT;
		bHorn : USINT;
		bLight : USINT;
		wCmdRet : UINT;
	END_STRUCT;
	IFmnMsgIn_Typ : 	STRUCT
		wCmd : UINT;
		wFunction_ID : UINT;
		wMsgNumber : UINT;
		wInstance : UINT;
		wMsgHistListSetOffset : UINT; (*Offset zum ersten Eintrag im originalen Ringbuffer.*)
		wMsgHistListClassSelect : UINT; (*Bitweise kodiert.*)
		wMsgHistListEventSelect : UINT; (*Eventnummer eintragen. 1..3. 0 - Alle anzeigen*)
		wMsgStatisticSelect : UINT; (*0 - *)
	END_STRUCT;
	IFmnMsgTrig_Typ : 	STRUCT
		xTrigPrevMsgHistListPage : BOOL;
		xTrigNextMsgHistListPage : BOOL;
		xMsgHistListPointToMin : BOOL;
		xRefreshHistList : BOOL;
		xSetHistListOffset : BOOL;
		xRefreshStatistic : BOOL;
	END_STRUCT;
	IFmnMsg_Typ : 	STRUCT
		In : IFmnMsgIn_Typ;
		Out : IFmnMsgOut_Typ;
		Trig : IFmnMsgTrig_Typ; (*Trigger werden von außen gesetzt und im Package zurückgesetzt*)
	END_STRUCT;
END_TYPE

(*Additional Status*)

TYPE
	mnMsgStatAdMsg_Typ : 	STRUCT
		dtMsgIntFaultChanged : DATE_AND_TIME;
		dtMsgExtFaultChanged : DATE_AND_TIME;
		dtMsgWarningChanged : DATE_AND_TIME;
		dtMsgInfoChanged : DATE_AND_TIME;
		dtMsgMaintChanged : DATE_AND_TIME;
		MsgCntFaultInt : USINT;
		MsgCntFaultExt : USINT;
		MsgCntWarning : USINT;
		MsgCntInformation : USINT;
		MsgCntMaintenance : USINT;
		bHorn : USINT;
		Reserve : ARRAY[0..1]OF USINT;
		MsgListFaultInt : ARRAY[0..MNMSG_MAX_MSGLIST]OF MsgList_Typ;
		MsgListFaultExt : ARRAY[0..MNMSG_MAX_MSGLIST]OF MsgList_Typ;
		MsgListWarning : ARRAY[0..MNMSG_MAX_MSGLIST]OF MsgList_Typ;
		MsgListInformation : ARRAY[0..MNMSG_MAX_MSGLIST]OF MsgList_Typ;
		MsgListMaintenance : ARRAY[0..MNMSG_MAX_MSGLIST]OF MsgList_Typ;
	END_STRUCT;
	mnMsgStatAd_Typ : 	STRUCT
		Msg : mnMsgStatAdMsg_Typ;
		sPkgVersion : STRING[10];
		xReady : BOOL;
	END_STRUCT;
END_TYPE

(*Parameter*)

TYPE
	mnMsgPar_Typ : 	STRUCT
		Mac : mnMsgParMac_Typ;
	END_STRUCT;
	mnMsgParMac_Typ : 	STRUCT
		wModeHorn : UINT;
		wTimeOnFault : UINT;
		wTimeOffFault : UINT;
		wTimeOnWarning : UINT;
		wTimeOffWarning : UINT;
	END_STRUCT;
END_TYPE
```

### Pkg_mnMsg.var - Package variables
```iecst
(********************************************************************
 * COPYRIGHT -- Microsoft
 ********************************************************************
 * Package: Pkg_mnMsg
 * File: Pkg_mnMsg.var
 * Author: hunholz, Subramaniam
 * Created: January 05, 2011
 * Changed: June 15, 2011
 ********************************************************************
 * Variables of package Pkg_mnMsg
 ********************************************************************)
(*Konstanten für Kommandos*)
VAR CONSTANT
	MNMSG_CMD_HORN_OFF : UINT := 1; (*Kommando, Horn aus*)
	MNMSG_CMD_ACK_FAULT : UINT := 2; (*Quittiere alle Störungen*)
	MNMSG_CMD_ACK_MAINT : UINT := 3; (*Quittiere alle Wartungen*)
	MNMSG_CMD_ACK : UINT := 4; (*Quittiere Einzelmeldung*)
	MNMSG_CMD_DEL_STAT : UINT := 5; (*Statistik löschen*)
	MNMSG_CMD_DEL_HIST : UINT := 6; (*Historie löschen*)
END_VAR
(*Kommandostati*)
VAR CONSTANT
	MNMSG_CMDSTAT_STATNOTREADY : UINT := 60000; (*Statistik ist nicht verfügbar*)
	MNMSG_CMDSTAT_HISTNOTREADY : UINT := 60001; (*Historie ist nicht verfügbar*)
	MNMSG_CMDSTAT_DELSTATFAILED : UINT := 60002; (*Statistik wurde nicht korrekt gelöscht*)
	MNMSG_CMDSTAT_DELHISTFAILED : UINT := 60003; (*Historie wurde nicht korrekt gelöscht*)
END_VAR
(*Modus der Hupe*)
VAR CONSTANT
	MNMSG_HORNMODE_OFF : UINT := 0;
	MNMSG_HORNMODE_ON : UINT := 1;
	MNMSG_HORNMODE_INTERV : UINT := 2;
END_VAR
(*Definition von Fehlern  *)
VAR CONSTANT
	MNMSG_MSG_NO_STATISTIC : UINT := 1000; (*Statistik ist fehlerhaft. Siehe Logbuch SPS.*)
	MNMSG_MSG_NO_HISTORY : UINT := 1003; (*Historie (Ringbuffer) ist fehlerhaft. Siehe Logbuch SPS.*)
	MNMSG_MSG_SYSTEMFAULT : UINT := 9999; (*Systemfehler Meldungsmanager*)
END_VAR
(*Sortiermodi für Meldungsstatistik*)
VAR CONSTANT
	MNMSG_STATMODE_CNT : UINT := 0; (*Die Meldungsstatistik soll nach Häufigkeit sortiert werden*)
	MNMSG_STATMODE_TIME : UINT := 1; (*Die Meldungsstatistik soll nach Dauer sortiert werden*)
END_VAR
(*Kommandschnittstelle Visualisierung *)
VAR
	mnMsgCmd : KG_Cmd_typ := (0);
	IFmnMsg : IFmnMsg_Typ := (0);
	mnMsgPar : mnMsgPar_Typ := (0);
	mnMsgStatAd : mnMsgStatAd_Typ;
END_VAR
(*Meldungsschnittstelle*)
VAR
	kgMsgStatus : ARRAY[0..MNMSG_MAX_IDX_KGMSGSTATUS] OF kgMsg_Status_Typ;
END_VAR
```

### Program Logical/Standard/Kanlink/KGFramework/Pkg_mnMsg/mnMsg (IEC) - Meldungsmanager
